// TwinCAT 3 PLC project HotdogMaker
// ProgramVersion: 3.1.4026.20
// libraries:
//   Tc2_ControllerToolbox, * (Beckhoff Automation GmbH)
//   Tc2_Standard, * (Beckhoff Automation GmbH)
//   Tc2_System, * (Beckhoff Automation GmbH)
// project tree:
//   GVLs/ GVL.TcGVL
//   / PlcTask.TcTTO
//   POUs/ MAIN.TcPOU
// real-time tasks:
//   TASK PlcTask: cycle T#10ms, priority 20, ADS port 350
// I/O:
//   DEVICE Device 1 (EtherCAT), AmsNetId 169.254.227.188.2.1
//     Term 1 (EK1100) [EK1100 EtherCAT Coupler (2A E-Bus)]
//       Term 2 (EL1018) [EL1018 8Ch. Dig. Input 24V, 10µs]
//       Term 3 (EL2008) [EL2008 8Ch. Dig. Output 24V, 0.5A]
//       Term 4 (EL3102) [EL3102 2Ch. Ana. Input +/-10V, Diff.]
//       Term 5 (EL2124) [EL2124 4Ch. Dig. Output 5V, 20mA]
//       Term 6 (EL9011) [EL9011 End Terminal]
// variable links:
//   HotdogMaker/HotdogMaker Instance <-> Device 1 (EtherCAT)/Term 1 (EK1100)/Term 3 (EL2008)
//     PlcTask Outputs/GVL.heaterElementEnable <-> Channel 2/Output
//   HotdogMaker/HotdogMaker Instance <-> Device 1 (EtherCAT)/Term 1 (EK1100)/Term 4 (EL3102)
//     PlcTask Inputs/GVL.temperatureSensor <-> AI Standard Channel 2/Value
//     PlcTask Inputs/GVL.temperatureSensorCopy <-> AI Standard Channel 1/Value

CONFIGURATION HotdogMaker
    RESOURCE PLC ON TwinCAT3
        TASK PlcTask(INTERVAL := T#10ms, PRIORITY := 20);
        PROGRAM MAIN WITH PlcTask : MAIN;
    END_RESOURCE
END_CONFIGURATION

// ---- GVLs/GVL.TcGVL
{attribute 'qualified_only'}
VAR_GLOBAL
	heaterElementEnable AT%Q* : BOOL := FALSE;
	temperatureSensorCopy AT%I* : INT := 0;
	temperatureSensor AT%I* : INT := 0;
END_VAR

// ---- POUs/MAIN.TcPOU
PROGRAM MAIN
VAR
	flagStartup: BOOL := FALSE;
	measuredTemperature : REAL := 0.0;
	K_GAIN : REAL := 0.025;
	B_OFFSET : REAL := 45;
	
	(*PI-Controller Parameter Struct*)
	PI_Ctrl_param 	  : ST_CTRL_PI_PARAMS; 

	(*PI-Controller*)
	fTargetTemperature : REAL := 200;
    fManSyncValue     : REAL  := 200;
	
	fOut 			  : REAL := 0;
    bSync             : BOOL;
    eMode             : E_CTRL_MODE := eCTRL_MODE_ACTIVE;
    bHold             : BOOL;
						
	PI_Ctrl 		  : FB_CTRl_Pi;
	
	(*PWM_Controller PWM*)
	PWM_Ctrl_param 	  : ST_CTRL_PWM_OUT_PARAMS;
	
	(*PWM_Controller*)
	PWM_Ctrl 		  : FB_CTRL_PWM_OUT;
END_VAR

IF flagStartup = FALSE THEN
	
	(*Fill PI-Ctrl - parameter struct*)
	PI_Ctrl_param.tCtrlCycleTime := T#10S;
	PI_Ctrl_param.tTaskCycleTime := T#1S;
	PI_Ctrl_param.tTn := T#160S;
	PI_Ctrl_param.fKp := 5.4;
	PI_Ctrl_param.fOutMinLimit := 0.0;
	PI_Ctrl_param.fOutMaxLimit := 200.0;
	
	(*Fill PWM-Ctrl - parameter struct*)
	PWM_Ctrl_param.tPWMPeriod := T#10S;
	PWM_Ctrl_param.tTaskCycleTime := T#1S;
	PWM_Ctrl_param.bInstantPWMUpdate := TRUE;
	
	(*End Startup procedure*)
	flagStartup := TRUE;		
END_IF
(*Raumptemperatur entspricht ca -1000 bei 20 Grad*)
(*Messung entspricht ca -1000 bei 20 Grad*)

GVL.heaterElementEnable := TRUE;

measuredTemperature := INT_TO_REAL(GVL.temperatureSensor) * K_GAIN + B_OFFSET;

(*Run PI-Ctrler*)
PI_Ctrl(
	stParams :=PI_Ctrl_param,
	fSetpointValue := fTargetTemperature,
	eMode := eMode,
	fActualValue := measuredTemperature,
	fManSyncValue := fManSyncValue,
	bHold := bHold,
	bSync  := bSync
);
fout := PI_Ctrl.fOut;
			
(*Run PWM-Ctrl*)
PWM_Ctrl(
	stParams := PWM_Ctrl_param,
	eMode := eCTRL_MODE_ACTIVE,
	fPwmInput := TO_LREAL(fout));
	
GVL.heaterElementEnable := PWM_Ctrl.bPwmOutBitPos;

END_PROGRAM
